// TwinCAT 3 PLC project Nepionic_Metrics_OTel
// Title: Nepionic_Metrics_OTel
// Company: Nepionic
// Author: Nepionic
// ProjectVersion: 0.1.0
// ProgramVersion: 3.1.4026.22
// libraries:
//   [Nepionic_Metrics], * (Nepionic)
//   Tc2_System, * (Beckhoff Automation GmbH)
//   Tc2_Utilities, * (Beckhoff Automation GmbH)
// project tree:
//   Lib/ OTelMetricCore.TcPOU, OTelMetricEntry.TcDUT, OTelMetricRing.TcDUT

// ---- Lib/OTelMetricEntry.TcDUT
// One slot in OtelMetricRing.
//
// Binary layout (672 bytes, little-endian — matches Go parser in adsbridge/ringbuf.go):
//
//   offset   0  ULINT   timestamp         Unix epoch nanoseconds
//   offset   8  UDINT   kind              0=Gauge 1=Counter 2=UpDownCounter
//   offset  12  UDINT   attr_count        Number of populated attrs (0..5)
//   offset  16  BYTE[128] name            STRING(127) null-terminated
//   offset 144  BYTE[32]  unit            STRING(31)  null-terminated
//   offset 176  LREAL   value             Metric value
//   offset 184  MetricAttribute[5]        5 x 96 bytes = 480 bytes
//                                           key STRING(31)=32 bytes
//                                           value STRING(63)=64 bytes
//   offset 664  BYTE[4]   _pad
//   offset 668  UDINT   sequence          ODD=being written, EVEN=committed (LAST field)
//   Total: 672 bytes
TYPE OTelMetricEntry :
STRUCT
	timestamp  : ULINT;
	kind       : UDINT;
	attr_count : UDINT;
	name       : STRING(127);
	unit       : STRING(31);
	value      : LREAL;
	attrs      : ARRAY[0..4] OF Nepionic_Metrics.MetricAttribute;
	_pad       : ARRAY[0..3] OF BYTE;
	sequence   : UDINT;
END_STRUCT
END_TYPE

// ---- Lib/OTelMetricRing.TcDUT
// Ring buffer header + 256-slot metric entry array.
// Exposed as an ADS symbol (e.g. OtelBridge.MetricRing) and read by the Go collector.
//
// Binary layout:
//   offset      0  UDINT  head          Monotonically increasing write counter
//   offset      4  UDINT  capacity      Number of slots = 256
//   offset      8  UDINT  overflow_cnt  Incremented when ring is full
//   offset     12  UDINT  _reserved
//   offset     16  BYTE[48] _cache_pad  Pad header to 64 bytes
//   offset     64  OtelMetricEntry[256] 256 x 672 bytes = 172032 bytes
//   Total: 172096 bytes
TYPE OTelMetricRing :
STRUCT
	head         : UDINT;
	capacity     : UDINT := 256;
	overflow_cnt : UDINT;
	_reserved    : UDINT;
	_cache_pad   : ARRAY[0..47] OF BYTE;
	entries      : ARRAY[0..255] OF OTelMetricEntry;
END_STRUCT
END_TYPE

// ---- Lib/OTelMetricCore.TcPOU
{attribute 'linkalways'}
{attribute 'no_explicit_call' := 'This FB is a CLASS and must be accessed using methods or properties'}
{attribute 'enable_dynamic_creation'}
/// OTel backend for Nepionic_Metrics.
/// Implements MetricCore by writing structured metric entries directly into an
/// OtelMetricRing that is exposed as an ADS symbol and consumed by the Go
/// otelcol-ads collector via the push_ring path.
///
/// Usage:
///   1. Declare an OtelMetricRing somewhere accessible via ADS (e.g. in a PROGRAM).
///   2. Set Ring := ADR(myMetricRing) before any Record calls.
///   3. Assign THIS^ to a Meter instance via meter.Core := THIS^.
FUNCTION_BLOCK PUBLIC OTelMetricCore IMPLEMENTS Nepionic_Metrics.MetricCore
VAR
	_ring : POINTER TO OTelMetricRing;
END_VAR

// No cyclic body — all logic is in methods.

METHOD PUBLIC Record : BOOL
VAR_INPUT
	name       : STRING(127);
	unit       : STRING(31);
	value      : LREAL;
	kind       : Nepionic_Metrics.MetricKind;
	attrs      : ARRAY[0..4] OF Nepionic_Metrics.MetricAttribute;
	attr_count : USINT;
END_VAR
VAR
	slot_idx : UDINT;
	expected_gen : UDINT;
	ft : Tc2_Utilities.T_FILETIME;
	ft_ulint : ULINT;
	i : USINT;
END_VAR
IF _ring = 0 THEN
	Record := FALSE;
	RETURN;
END_IF

slot_idx     := _ring^.head MOD _ring^.capacity;
expected_gen := (_ring^.head / _ring^.capacity + 1) * 2;

// Mark slot as being written (ODD sequence = write in progress)
_ring^.entries[slot_idx].sequence := expected_gen - 1;

// Capture timestamp — Windows FILETIME to Unix nanoseconds
//ft := Tc2_Utilities.F_GetSystemTime();
ft_ulint := Tc2_Utilities.F_GetSystemTime(); //SHL(DWORD_TO_ULINT(ft.dwHighDateTime), 32) OR DWORD_TO_ULINT(ft.dwLowDateTime);
_ring^.entries[slot_idx].timestamp := (ft_ulint - 116444736000000000) * 100;

_ring^.entries[slot_idx].kind       := TO_UDINT(kind);
_ring^.entries[slot_idx].name       := name;
_ring^.entries[slot_idx].unit       := unit;
_ring^.entries[slot_idx].value      := value;
_ring^.entries[slot_idx].attr_count := USINT_TO_UDINT(attr_count);

FOR i := 0 TO 4 DO
	_ring^.entries[slot_idx].attrs[i] := attrs[i];
END_FOR

// Increment overflow counter each time the write pointer wraps back to slot 0.
// slot_idx = 0 and head > 0 means we are about to overwrite the oldest entries.
IF slot_idx = 0 AND _ring^.head > 0 THEN
	_ring^.overflow_cnt := _ring^.overflow_cnt + 1;
END_IF

// Mark slot as committed (EVEN sequence = ready to read)
_ring^.entries[slot_idx].sequence := expected_gen;

_ring^.head := _ring^.head + 1;
Record := TRUE;
END_METHOD

{attribute 'monitoring' := 'call'}
PROPERTY PUBLIC Ring : POINTER TO OTelMetricRing
GET
Ring := _ring;
END_GET
SET
_ring := Ring;
END_SET
END_PROPERTY

END_FUNCTION_BLOCK
